// TIA Portal project "Proyecto" (V16)

(* hardware
DEVICE "S71500/ET200MP station_1"  S7-1500 station
   slot 0: "Perfil soporte_0"  Rack  6ES7 590-1***0-0AA0
   slot 1: "PLC_1"  CPU 1511-1 PN  6ES7 511-1AK01-0AB0  V2.8
      slot 3: "Display de la CPU_1"  6ES7591-1AA00-0AA0
      slot 32768: "Interfaz PROFINET_1"  X1
         slot 32769: "Puerto_1"  X1 P1
         slot 32770: "Puerto_2"  X1 P2
      slot 34817: "Virtual CP interface port_1"  Virtual CP interface port  Virtual CP interface port
DEVICE "S71500/ET200MP station_2"  S7-1500 station
   slot 0: "Perfil soporte_0"  Rack  6ES7 590-1***0-0AA0
   slot 1: "PLC_2"  CPU 1511-1 PN  6ES7 511-1AK01-0AB0  V2.8
      slot 3: "Display de la CPU_1"  6ES7591-1AA00-0AA0
      slot 32768: "Interfaz PROFINET_1"  X1
         slot 32769: "Puerto_1"  X1 P1
         slot 32770: "Puerto_2"  X1 P2
      slot 34817: "Virtual CP interface port_1"  Virtual CP interface port  Virtual CP interface port
*)

// ===== PLC "PLC_1"  CPU 1511-1 PN =====

VAR_GLOBAL   // PLC tag table "Tabla de variables estándar"
   "System_Byte" AT %MB1 : Byte;
   "FirstScan" AT %M1.0 : Bool;
   "DiagStatusUpdate" AT %M1.1 : Bool;
   "AlwaysTRUE" AT %M1.2 : Bool;
   "AlwaysFALSE" AT %M1.3 : Bool;
   "Clock_Byte" AT %MB0 : Byte;
   "Clock_10Hz" AT %M0.0 : Bool;
   "Clock_5Hz" AT %M0.1 : Bool;
   "Clock_2.5Hz" AT %M0.2 : Bool;
   "Clock_2Hz" AT %M0.3 : Bool;
   "Clock_1.25Hz" AT %M0.4 : Bool;
   "Clock_1Hz" AT %M0.5 : Bool;
   "Clock_0.625Hz" AT %M0.6 : Bool;
   "Clock_0.5Hz" AT %M0.7 : Bool;
END_VAR

DATA_BLOCK "DataLogPLC1Maestro"   // DB1
{ S7_Optimized_Access := 'FALSE' }
VERSION : 0.1
   VAR
      Variable1 : Real := 0.55;
      SetPoint : Int := 5;
   END_VAR
BEGIN
END_DATA_BLOCK

DATA_BLOCK "ProduccionPLC_Campo"   // DB4
{ S7_Optimized_Access := 'FALSE' }
VERSION : 0.1
   VAR
      Produccion : Array[1..7] of Real;
      EstadoMaquina : Array[1..2] of Bool;
   END_VAR
BEGIN
END_DATA_BLOCK

DATA_BLOCK "EnvioVariables"   // DB5
{ S7_Optimized_Access := 'FALSE' }
VERSION : 0.1
   VAR
      Variables : Array[1..8] of Bool;
   END_VAR
BEGIN
   Variables[1] := TRUE;
   Variables[2] := TRUE;
END_DATA_BLOCK

// folder: System blocks/Program resources

DATA_BLOCK "PLC_1_Receive_DB"   // DB2
{ S7_Optimized_Access := 'TRUE' }
AUTHOR : SIMATIC
FAMILY : MC7Plus
NAME : IP_RFC
VERSION : 1.0
// stored: InstanceOfName TCON_IP_RFC
"TCON_IP_RFC"
BEGIN
   ID := 1;
   InterfaceId := 64;
   LocalTSelector.TSel[1] := B#16#E0;
   LocalTSelector.TSel[2] := B#16#01;
   LocalTSelector.TSel[3] := B#16#49;
   LocalTSelector.TSel[4] := B#16#53;
   LocalTSelector.TSel[5] := B#16#4F;
   LocalTSelector.TSel[6] := B#16#6F;
   LocalTSelector.TSel[7] := B#16#6E;
   LocalTSelector.TSel[8] := B#16#54;
   LocalTSelector.TSel[9] := B#16#43;
   LocalTSelector.TSel[10] := B#16#50;
   LocalTSelector.TSel[11] := B#16#2D;
   LocalTSelector.TSel[12] := B#16#31;
   LocalTSelector.TSelLength := 12;
   RemoteTSelector.TSel[1] := B#16#E0;
   RemoteTSelector.TSel[2] := B#16#01;
   RemoteTSelector.TSel[3] := B#16#49;
   RemoteTSelector.TSel[4] := B#16#53;
   RemoteTSelector.TSel[5] := B#16#4F;
   RemoteTSelector.TSel[6] := B#16#6F;
   RemoteTSelector.TSel[7] := B#16#6E;
   RemoteTSelector.TSel[8] := B#16#54;
   RemoteTSelector.TSel[9] := B#16#43;
   RemoteTSelector.TSel[10] := B#16#50;
   RemoteTSelector.TSel[11] := B#16#2D;
   RemoteTSelector.TSel[12] := B#16#31;
   RemoteTSelector.TSelLength := 12;
   RemoteAddress.ADDR[1] := 192;
   RemoteAddress.ADDR[2] := 168;
   RemoteAddress.ADDR[4] := 41;
END_DATA_BLOCK

DATA_BLOCK "PLC_1_Send_DB"   // DB7
{ S7_Optimized_Access := 'TRUE' }
AUTHOR : SIMATIC
FAMILY : MC7Plus
NAME : IP_RFC
VERSION : 1.0
// stored: InstanceOfName TCON_IP_RFC
"TCON_IP_RFC"
BEGIN
   ID := 2;
   InterfaceId := 64;
   RemoteTSelector.TSel[1] := B#16#50;
   RemoteTSelector.TSel[2] := B#16#4C;
   RemoteTSelector.TSel[3] := B#16#43;
   RemoteTSelector.TSel[4] := B#16#32;
   RemoteTSelector.TSel[5] := B#16#5F;
   RemoteTSelector.TSel[6] := B#16#52;
   RemoteTSelector.TSel[7] := B#16#45;
   RemoteTSelector.TSel[8] := B#16#43;
   RemoteTSelector.TSel[9] := B#16#49;
   RemoteTSelector.TSel[10] := B#16#42;
   RemoteTSelector.TSel[11] := B#16#45;
   RemoteTSelector.TSelLength := 11;
   LocalTSelector.TSel[1] := B#16#50;
   LocalTSelector.TSel[2] := B#16#4C;
   LocalTSelector.TSel[3] := B#16#43;
   LocalTSelector.TSel[4] := B#16#31;
   LocalTSelector.TSel[5] := B#16#5F;
   LocalTSelector.TSel[6] := B#16#45;
   LocalTSelector.TSel[7] := B#16#4E;
   LocalTSelector.TSel[8] := B#16#56;
   LocalTSelector.TSel[9] := B#16#49;
   LocalTSelector.TSel[10] := B#16#41;
   LocalTSelector.TSelLength := 10;
   RemoteAddress.ADDR[1] := 192;
   RemoteAddress.ADDR[2] := 168;
   RemoteAddress.ADDR[4] := 41;
END_DATA_BLOCK

DATA_BLOCK "PLC_1_Receive_DB_1"   // DB8
{ S7_Optimized_Access := 'TRUE' }
AUTHOR : SIMATIC
FAMILY : MC7Plus
NAME : IP_RFC
VERSION : 1.0
// stored: InstanceOfName TCON_IP_RFC
"TCON_IP_RFC"
BEGIN
   ID := 3;
   InterfaceId := 64;
   LocalTSelector.TSel[1] := B#16#E0;
   LocalTSelector.TSel[2] := B#16#01;
   LocalTSelector.TSel[3] := B#16#49;
   LocalTSelector.TSel[4] := B#16#53;
   LocalTSelector.TSel[5] := B#16#4F;
   LocalTSelector.TSel[6] := B#16#6F;
   LocalTSelector.TSel[7] := B#16#6E;
   LocalTSelector.TSel[8] := B#16#54;
   LocalTSelector.TSel[9] := B#16#43;
   LocalTSelector.TSel[10] := B#16#50;
   LocalTSelector.TSel[11] := B#16#2D;
   LocalTSelector.TSel[12] := B#16#31;
   LocalTSelector.TSelLength := 12;
   RemoteTSelector.TSel[1] := B#16#E0;
   RemoteTSelector.TSel[2] := B#16#01;
   RemoteTSelector.TSel[3] := B#16#49;
   RemoteTSelector.TSel[4] := B#16#53;
   RemoteTSelector.TSel[5] := B#16#4F;
   RemoteTSelector.TSel[6] := B#16#6F;
   RemoteTSelector.TSel[7] := B#16#6E;
   RemoteTSelector.TSel[8] := B#16#54;
   RemoteTSelector.TSel[9] := B#16#43;
   RemoteTSelector.TSel[10] := B#16#50;
   RemoteTSelector.TSel[11] := B#16#2D;
   RemoteTSelector.TSel[12] := B#16#31;
   RemoteTSelector.TSelLength := 12;
   RemoteAddress.ADDR[1] := 192;
   RemoteAddress.ADDR[2] := 168;
   RemoteAddress.ADDR[4] := 41;
END_DATA_BLOCK

// folder: (top level)

FUNCTION "Generador_incremental" : Void   // FC1, SCL
{ S7_Optimized_Access := 'TRUE' }
VERSION : 0.1
   VAR_INPUT
      minimo : Real;
      maximo : Real;
      incremento : Real;
   END_VAR
   VAR_IN_OUT
      aleatorio : Real;
   END_VAR
BEGIN
   REGION Ajustar el valor minimo
       IF #aleatorio < #minimo THEN
           #aleatorio := #minimo;
       END_IF;
   END_REGION

   REGION Generador Incremental
       IF #aleatorio < #maximo THEN
           #aleatorio := #aleatorio + #incremento;
       ELSE
           #aleatorio := #minimo;
       END_IF;
   END_REGION
END_FUNCTION

FUNCTION "RecibirProduccion" : Void   // FC2, LAD
{ S7_Optimized_Access := 'TRUE' }
VERSION : 0.1
BEGIN

REGION Network 1
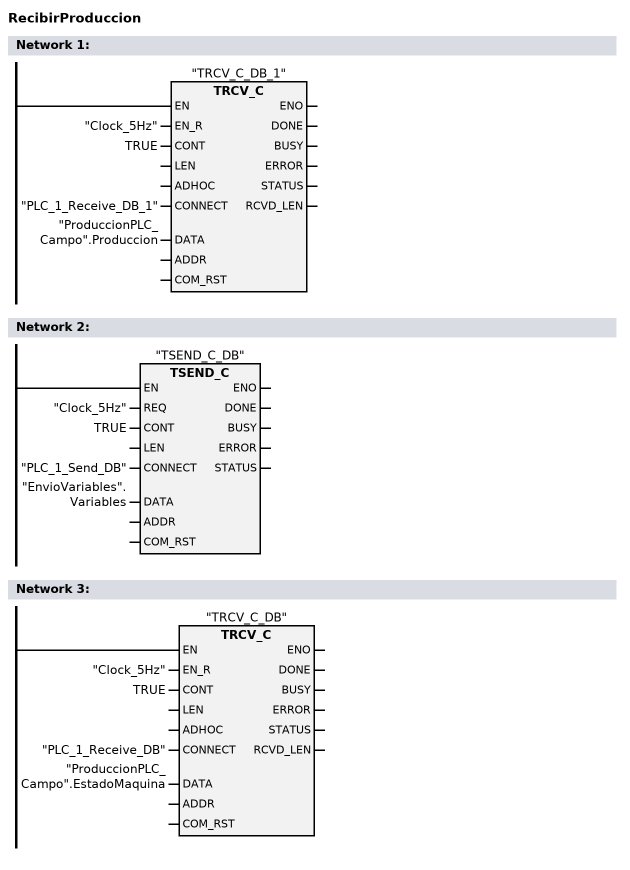
   "TRCV_C_DB_1"(EN_R := "Clock_5Hz",   // TRCV_C
                 CONT := TRUE,
                 CONNECT := "PLC_1_Receive_DB_1",
                 DATA := "ProduccionPLC_Campo".Produccion);
END_REGION

REGION Network 2
   "TSEND_C_DB"(REQ := "Clock_5Hz",   // TSEND_C
                CONT := TRUE,
                CONNECT := "PLC_1_Send_DB",
                DATA := "EnvioVariables".Variables);
END_REGION

REGION Network 3
   "TRCV_C_DB"(EN_R := "Clock_5Hz",   // TRCV_C
               CONT := TRUE,
               CONNECT := "PLC_1_Receive_DB",
               DATA := "ProduccionPLC_Campo".EstadoMaquina);
END_REGION
END_FUNCTION

ORGANIZATION_BLOCK "Main"   // OB1, LAD, ProgramCycle
TITLE = "Main Program Sweep (Cycle)"
{ S7_Optimized_Access := 'TRUE' }
VERSION : 0.1
   VAR_INPUT
      Initial_Call : Bool;   // Initial call of this OB
      Remanence : Bool;   // =True, if remanent data are available
   END_VAR
BEGIN

REGION Network 1
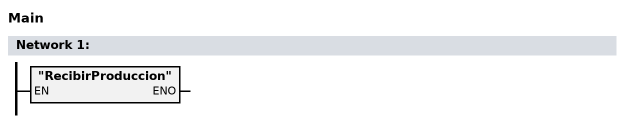
   RUNG wire#powerrail
      "RecibirProduccion"()
   END_RUNG
   // the same network as SCL:
   "RecibirProduccion"();
END_REGION
END_ORGANIZATION_BLOCK

// folder: LGF/4 Math operations

FUNCTION "LGF_RandomRange_Real" : Real   // FC10014, SCL
TITLE = LGF_RandomRange_Real
{ S7_Optimized_Access := 'TRUE' }
AUTHOR : Siemens_Digital_Industries
FAMILY : LGF
NAME : LGF_RandomRange_Real
// This function generates a random value in defined limits with each call.  
// The random number has the data type Real in the specified range.
// Diese Funktion generiert bei jedem Aufruf einen zufälligen Wert zwischen einem definierten Max- und Minwert.  
// Die Zufallszahl hat den Datentyp Real im spezifiziertem Wertebereich.
   VAR_INPUT
      minValue : Real;   // Minimalwert der für den Wertebereich der Zufallszahl - Untergrenze / Minimum value of the range of the random number - lower border
      maxValue : Real;   // Maximalwert der für den Wertebereich der Zufallszahl - Obergrenze / Maximum value of the range of the random number - upper border
   END_VAR
   VAR_OUTPUT
      error : Bool;   // FALSE: No error TRUE: An error occurred during the execution of the FB / FALSE: Kein Fehler TRUE: Während der Ausführung des FB ist ein Fehler aufgetreten
      status : Word;   // 16#0000-16#7FFF: Status of the FB 16#8000-16#FFFF: Error identification (see following Table) / 16#0000-16#7FFF: Status des FB 16#8000-16#FFFF: Fehleridentifikation (siehe folgende Tabelle)
      subfunctionStatus : Word;   // Status or return value of called FB's, FC's and system blocks / Status oder Rückgabewert von aufgerufenen FB's / FC's und Systemfunktionen
   END_VAR
   VAR_TEMP
      tempTime : DTL;   // Temp memory for System time / Temp variable für System Zeit
      tempNanoSecondInDWord : DWord;   // Temp UDInt converted to DWord for access to individual bytes / Temp UDInt konvertiert nach Dword für den Zufriff per Slice auf die Bytes
      tempTimeStatus : Word;   // Temp status of the instruction `RD_SYS_T` / Temp Status der Systemfunktion `RD_SYS_T`
      tempRandomValue : DWord;   // Temp Random startvalue / Temp Zufallswert als Startwert
      tempNormReal : Real;   // Temp normalized Real value (0.0 - 1.0) / Temp Normalisierer Realwert (0.0 - 1.0)
   END_VAR
   // Ret_Val : Random Real number in the predefined range / Zufallszahl vom Datentyp Real im definierten Wertebereich
   VAR CONSTANT
      ZERO : Real := 0.0;   // Zero / 0.0 - value in case of error / Null / 0.0 - Rückgabewert im Fehlerfall
      MAX_UDINT : UDInt := 4294967295;   // Maximum UDInt datatype / Maximalwert eines UDInt Datentype
      SUB_STATUS_NO_ERROR : Word := 16#0000;   // Status: sub function call ends without error / Status: Unterfunktionsaufruf ohne Fehler beendet
      STATUS_FINISHED_NO_ERROR : Word := 16#0000;   // Execution finished without errors / Abarbeitung ohne Fehler beendet
      ERR_MAX_LESS_MIN : Word := 16#8200;   // Error: The ranges specified are wrong: `minValue` is greater than `maxValue` / Fehler: Der spezifizierte Wetebereich is fehlerhaft: `minValue` ist größer als `maxValue`
      ERR_RD_SYS_T : Word := 16#8600;   // Error in `RD_SYS_T` command - check `subFunctionStatus` code / Fehler in Anweisung `RD_SYS_T` - weitere infos in `subFunctionStatus`
   END_VAR
BEGIN
   REGION Block info header
     //=============================================================================
     // SIEMENS AG / (c)Copyright 2017
     //-----------------------------------------------------------------------------
     // Title:            LGF_RandomRange_Real
     // Comment/Function: This function generates random numbers in defined limits (Datatype Real)
     // Library/Family:   LGF(Library General Functions)
     // Author:           Siemens Digital Industry Support
     // Tested with:      S7-PLCSIM Advanced V2.0 SP1
     // Engineering:      TIA Portal V15 Update 2
     // Restrictions:     ENO disabled - error handling done by error and status
     // Requirements:     PLC (S7-1200 / S7-1500)
     //-------------------------------------------------------------------------------
     // Change log table:
     // Version  | Date       | Expert in charge       | Changes applied
     //----------|------------|------------------------|------------------------------
     // 01.00.00 19.08.2015  Siemens Industry Online Support
     //                      First released version
     // 01.00.01 02.01.2017  Siemens Industry Online Support
     //                      Upgrade: TIA Portal V14 Update 1
     // 01.00.02 02.03.2017  Siemens Industry Online Support
     //                      Bugfix: FC number
     // 01.00.03 17.08.2018  Siemens Industry Online Support
     //                      Upgrade: TIA V15 Update 2
     // 01.00.04 23.11.2018  Siemens Industry Online Support
     //                      Upgrade: TIA V15.1
     // 01.01.00 13.11.2019  Simatic Systems Support
     //                      Renamed from "LGF_RandomReal" to "LGF_RandomRange_Real"
     //                      Regions, comments and constants are added
     // 03.00.00 23.04.2020  Simatic Systems Support
     //                      Set version to V3.0.0, harmonize the version of the whole library
     // 03.00.01 04.02.2021  Simatic Systems Support
     //                      Insert documentation
     //=============================================================================
   END_REGION Block info header

   REGION DESCRIPTION
     (/*Note
   :    The status of called commands is output in `subFunctionStatus`. In this case, the output value in `status` indicates which command caused the error. In this case, refer to the TIA Portal Online Help section for information on the respective commands.

   The block generates random values that are between the specified `minValue` and the `maxValue`. This random value is output via the `Ret_Val`.

   The random value is formed from the nanoseconds of the current system time of the CPU. The byte order of this value is inverted and then converted to a floating point.
   Hinweis
   :    In `subFunctionStatus` wird der Status von aufgerufenen Anweisungen ausgegeben. Der Ausgangswert in `status` gibt in diesem Fall an, welche Anweisung den Fehler verursacht hat. Holen Sie sich in diesem Fall die Informationen aus der TIA Portal Online Hilfe zu den jeweiligen Anweisungen.

   Der Baustein generiert zufällige Werte, die zwischen dem angegebenen `minValue`-Wert und `maxValue`-Wert liegen. Dieser zufällige Wert wird über den `Ret_Val` ausgegeben.

   Der Zufallswert wird aus den Nanosekunden der aktuellen Systemzeit der CPU gebildet. Dabei wird die Bytereihenfolge dieses Wertes invertiert und anschließend in eine Gleitkommazahl ungewandelt.*/)
   END_REGION DESCRIPTION

   REGION Validation
     // Check if the maximal Value is less than the minimal value
     IF (#minValue > #maxValue) THEN
       #error := true;
       #status := #ERR_MAX_LESS_MIN;
       #subfunctionStatus := #SUB_STATUS_NO_ERROR;
       #LGF_RandomRange_Real := #ZERO;
       RETURN;
     END_IF;

     // Read system time
     #tempTimeStatus := INT_TO_WORD(RD_SYS_T(#tempTime));

     // Check return variable for error
     IF (#tempTimeStatus <> #SUB_STATUS_NO_ERROR) THEN
       #error := true;
       #status := #ERR_RD_SYS_T;
       #subfunctionStatus := #tempTimeStatus;
       #LGF_RandomRange_Real := #ZERO;
       RETURN;
     END_IF;
   END_REGION

   REGION Calculating random number
     // Converting to double word so individual bytes can be addressed
     #tempNanoSecondInDWord := UDINT_TO_DWORD(#tempTime.NANOSECOND);

     // Calculate a random-start-value depending on the time
     #tempRandomValue.%B3 := #tempNanoSecondInDWord.%B0;
     #tempRandomValue.%B2 := #tempNanoSecondInDWord.%B1;
     #tempRandomValue.%B1 := #tempNanoSecondInDWord.%B2;
     #tempRandomValue.%B0 := #tempNanoSecondInDWord.%B3;

     // Norm the calculated random number: 0.0 <= #tempNormReal <= 1.0
     #tempNormReal := UDINT_TO_REAL(DWORD_TO_UDINT(#tempRandomValue)) / UDINT_TO_REAL(#MAX_UDINT);

     // Scale the tempNormReal to be in the range of maxValue and minValue
     #LGF_RandomRange_Real := ((#tempNormReal * (#maxValue - #minValue) + (#minValue)));

     #error := false;
     #status := #STATUS_FINISHED_NO_ERROR;
     #subfunctionStatus := #SUB_STATUS_NO_ERROR;
     // ENO mechanism is not used
     ENO := TRUE;
   END_REGION
END_FUNCTION

// ===== PLC "PLC_2"  CPU 1511-1 PN =====

VAR_GLOBAL   // PLC tag table "Tabla de variables estándar"
   "System_Byte" AT %MB1 : Byte;
   "FirstScan" AT %M1.0 : Bool;
   "DiagStatusUpdate" AT %M1.1 : Bool;
   "AlwaysTRUE" AT %M1.2 : Bool;
   "AlwaysFALSE" AT %M1.3 : Bool;
   "Clock_Byte" AT %MB0 : Byte;
   "Clock_10Hz" AT %M0.0 : Bool;
   "Clock_5Hz" AT %M0.1 : Bool;
   "Clock_2.5Hz" AT %M0.2 : Bool;
   "Clock_2Hz" AT %M0.3 : Bool;
   "Clock_1.25Hz" AT %M0.4 : Bool;
   "Clock_1Hz" AT %M0.5 : Bool;
   "Clock_0.625Hz" AT %M0.6 : Bool;
   "Clock_0.5Hz" AT %M0.7 : Bool;
   "Start" AT %I1.2 : Bool;
   "PASO0" AT %M10.3 : Bool;
   "PASO1" AT %M10.4 : Bool;
   "PASO2" AT %M10.5 : Bool;
   "PASO3" AT %M10.6 : Bool;
   "PASO4" AT %M10.7 : Bool;
   "PASO5" AT %M11.0 : Bool;
   "PASO6" AT %M11.1 : Bool;
   "PASO7" AT %M11.2 : Bool;
   "PASO8" AT %M11.3 : Bool;
   "PASO9" AT %M11.4 : Bool;
   "Motor_bases" AT %Q0.3 : Bool;
   "Motor_tapas" AT %Q0.6 : Bool;
   "Detector_bases" AT %I0.3 : Bool;
   "Detector_tapas" AT %I0.6 : Bool;
   "Presionar_bases" AT %Q0.4 : Bool;
   "Presionar_tapas" AT %Q0.7 : Bool;
   "MoverZ" AT %Q0.1 : Bool;
   "MoverX" AT %Q0.0 : Bool;
   "Agarrar" AT %Q0.2 : Bool;
   "MoviendoseZ" AT %I0.1 : Bool;
   "ItemDetectado" AT %I0.2 : Bool;
   "MoviendoseX" AT %I0.0 : Bool;
   "Base_posicionada" AT %I0.4 : Bool;
   "Tapa_posicionada" AT %I0.7 : Bool;
   "PASO10" AT %M11.5 : Bool;
   "PASO11" AT %M12.0 : Bool;
   "PASO12" AT %M12.1 : Bool;
   "PASO13" AT %M12.2 : Bool;
   "PASO14" AT %M12.3 : Bool;
   "PASO15" AT %M12.4 : Bool;
   "PASO16" AT %M12.5 : Bool;
   "PASO17" AT %M12.6 : Bool;
   "PASO18" AT %M12.7 : Bool;
   "Libera_base" AT %Q1.0 : Bool;
   "Saliendo" AT %I1.1 : Bool;
   "PASO9_INTER" AT %M2.0 : Bool;
   "PASO2_INTER" AT %M2.1 : Bool;
   "PASO2_INTER2" AT %M2.2 : Bool;
   "Done" AT %M2.3 : Bool;
   "EmisorBases" AT %Q1.4 : Bool;
   "EmisorTapas" AT %Q1.5 : Bool;
   "SP_Cajas" AT %MW4 : Int;
   "SP_CajasAUX" AT %MW6 : Int;
   "RESET_COUNTER" AT %M2.4 : Bool;
   "PASO9_INTER2" AT %M2.5 : Bool;
   "SetPointInterno" AT %MW8 : Int;
   "Stop" AT %I1.4 : Bool;
   "AUX1" AT %M2.6 : Bool;
   "AUX2" AT %M2.7 : Bool;
   "AUX3" AT %M3.0 : Bool;
   "SET DETEC" AT %M3.1 : Bool;
   "Sensor tapa" AT %ID100 : DInt;
   "Sensor base" AT %ID104 : DInt;
   "Reset" AT %I1.3 : Bool;
   "Emergency stop" AT %I1.5 : Bool;
   "RESET_DONE" AT %M3.2 : Bool;
   "TiempoMinutos" AT %MD14 : Real;
   "FactoryRunning" AT %I1.7 : Bool;
   "TiempoTotal" AT %MD18 : Real;
   "Div1" AT %MD22 : Real;
END_VAR

DATA_BLOCK "Datalog"   // DB1
{ S7_Optimized_Access := 'FALSE' }
VERSION : 0.1
   VAR
      Variable1 : Real;
      SetPoint : Int := 4;
   END_VAR
BEGIN
END_DATA_BLOCK

DATA_BLOCK "Envio_Estados"   // DB12
{ S7_Optimized_Access := 'TRUE' }
VERSION : 0.1
   VAR
      Parametros : Array[1..7] of Real;
      EstadoMaquina : Array[1..2] of Bool;
   END_VAR
BEGIN
END_DATA_BLOCK

DATA_BLOCK "RecepcionVariables"   // DB17
{ S7_Optimized_Access := 'TRUE' }
VERSION : 0.1
   VAR
      Variables : Array[1..8] of Bool;
   END_VAR
BEGIN
END_DATA_BLOCK

// folder: System blocks/Program resources

DATA_BLOCK "IEC_Timer_0_DB"   // DB2
{ S7_Optimized_Access := 'TRUE' }
AUTHOR : Simatic
FAMILY : IEC
NAME : IEC_TMR
VERSION : 1.0
// stored: InstanceOfName IEC_TIMER
"IEC_TIMER"
BEGIN
END_DATA_BLOCK

DATA_BLOCK "IEC_Timer_0_DB_1"   // DB3
{ S7_Optimized_Access := 'TRUE' }
AUTHOR : Simatic
FAMILY : IEC
NAME : IEC_TMR
VERSION : 1.0
// stored: InstanceOfName IEC_TIMER
"IEC_TIMER"
BEGIN
END_DATA_BLOCK

DATA_BLOCK "IEC_Timer_0_DB_2"   // DB4
{ S7_Optimized_Access := 'TRUE' }
AUTHOR : Simatic
FAMILY : IEC
NAME : IEC_TMR
VERSION : 1.0
// stored: InstanceOfName IEC_TIMER
"IEC_TIMER"
BEGIN
END_DATA_BLOCK

DATA_BLOCK "IEC_Timer_0_DB_3"   // DB5
{ S7_Optimized_Access := 'TRUE' }
AUTHOR : Simatic
FAMILY : IEC
NAME : IEC_TMR
VERSION : 1.0
// stored: InstanceOfName IEC_TIMER
"IEC_TIMER"
BEGIN
END_DATA_BLOCK

DATA_BLOCK "IEC_Timer_0_DB_4"   // DB6
{ S7_Optimized_Access := 'TRUE' }
AUTHOR : Simatic
FAMILY : IEC
NAME : IEC_TMR
VERSION : 1.0
// stored: InstanceOfName IEC_TIMER
"IEC_TIMER"
BEGIN
END_DATA_BLOCK

DATA_BLOCK "IEC_Timer_0_DB_5"   // DB7
{ S7_Optimized_Access := 'TRUE' }
AUTHOR : Simatic
FAMILY : IEC
NAME : IEC_TMR
VERSION : 1.0
// stored: InstanceOfName IEC_TIMER
"IEC_TIMER"
BEGIN
END_DATA_BLOCK

DATA_BLOCK "IEC_Timer_0_DB_6"   // DB8
{ S7_Optimized_Access := 'TRUE' }
AUTHOR : Simatic
FAMILY : IEC
NAME : IEC_TMR
VERSION : 1.0
// stored: InstanceOfName IEC_TIMER
"IEC_TIMER"
BEGIN
END_DATA_BLOCK

DATA_BLOCK "IEC_Counter_0_DB"   // DB9
{ S7_Optimized_Access := 'TRUE' }
AUTHOR : Simatic
FAMILY : IEC
NAME : CNTR
VERSION : 1.0
// stored: InstanceOfName IEC_COUNTER
"IEC_COUNTER"
BEGIN
END_DATA_BLOCK

DATA_BLOCK "IEC_Timer_0_DB_8"   // DB10
{ S7_Optimized_Access := 'TRUE' }
AUTHOR : Simatic
FAMILY : IEC
NAME : IEC_TMR
VERSION : 1.0
// stored: InstanceOfName IEC_TIMER
"IEC_TIMER"
BEGIN
END_DATA_BLOCK

DATA_BLOCK "IEC_Timer_0_DB_7"   // DB11
{ S7_Optimized_Access := 'TRUE' }
AUTHOR : Simatic
FAMILY : IEC
NAME : IEC_TMR
VERSION : 1.0
// stored: InstanceOfName IEC_TIMER
"IEC_TIMER"
BEGIN
END_DATA_BLOCK

DATA_BLOCK "PLC_2_Send_DB"   // DB15
{ S7_Optimized_Access := 'TRUE' }
AUTHOR : SIMATIC
FAMILY : MC7Plus
NAME : IP_RFC
VERSION : 1.0
// stored: InstanceOfName TCON_IP_RFC
"TCON_IP_RFC"
BEGIN
   ID := 1;
   ActiveEstablished := true;
   InterfaceId := 64;
   RemoteAddress.ADDR[1] := 192;
   RemoteAddress.ADDR[2] := 168;
   RemoteAddress.ADDR[4] := 21;
   LocalTSelector.TSel[1] := B#16#E0;
   LocalTSelector.TSel[2] := B#16#01;
   LocalTSelector.TSel[3] := B#16#49;
   LocalTSelector.TSel[4] := B#16#53;
   LocalTSelector.TSel[5] := B#16#4F;
   LocalTSelector.TSel[6] := B#16#6F;
   LocalTSelector.TSel[7] := B#16#6E;
   LocalTSelector.TSel[8] := B#16#54;
   LocalTSelector.TSel[9] := B#16#43;
   LocalTSelector.TSel[10] := B#16#50;
   LocalTSelector.TSel[11] := B#16#2D;
   LocalTSelector.TSel[12] := B#16#31;
   LocalTSelector.TSelLength := 12;
   RemoteTSelector.TSel[1] := B#16#E0;
   RemoteTSelector.TSel[2] := B#16#01;
   RemoteTSelector.TSel[3] := B#16#49;
   RemoteTSelector.TSel[4] := B#16#53;
   RemoteTSelector.TSel[5] := B#16#4F;
   RemoteTSelector.TSel[6] := B#16#6F;
   RemoteTSelector.TSel[7] := B#16#6E;
   RemoteTSelector.TSel[8] := B#16#54;
   RemoteTSelector.TSel[9] := B#16#43;
   RemoteTSelector.TSel[10] := B#16#50;
   RemoteTSelector.TSel[11] := B#16#2D;
   RemoteTSelector.TSel[12] := B#16#31;
   RemoteTSelector.TSelLength := 12;
END_DATA_BLOCK

DATA_BLOCK "PLC_2_Receive_DB"   // DB16
{ S7_Optimized_Access := 'TRUE' }
AUTHOR : SIMATIC
FAMILY : MC7Plus
NAME : IP_RFC
VERSION : 1.0
// stored: InstanceOfName TCON_IP_RFC
"TCON_IP_RFC"
BEGIN
   ID := 2;
   ActiveEstablished := true;
   InterfaceId := 64;
   RemoteAddress.ADDR[1] := 192;
   RemoteAddress.ADDR[2] := 168;
   RemoteAddress.ADDR[4] := 21;
   LocalTSelector.TSel[1] := B#16#50;
   LocalTSelector.TSel[2] := B#16#4C;
   LocalTSelector.TSel[3] := B#16#43;
   LocalTSelector.TSel[4] := B#16#32;
   LocalTSelector.TSel[5] := B#16#5F;
   LocalTSelector.TSel[6] := B#16#52;
   LocalTSelector.TSel[7] := B#16#45;
   LocalTSelector.TSel[8] := B#16#43;
   LocalTSelector.TSel[9] := B#16#49;
   LocalTSelector.TSel[10] := B#16#42;
   LocalTSelector.TSel[11] := B#16#45;
   LocalTSelector.TSelLength := 11;
   RemoteTSelector.TSel[1] := B#16#50;
   RemoteTSelector.TSel[2] := B#16#4C;
   RemoteTSelector.TSel[3] := B#16#43;
   RemoteTSelector.TSel[4] := B#16#31;
   RemoteTSelector.TSel[5] := B#16#5F;
   RemoteTSelector.TSel[6] := B#16#45;
   RemoteTSelector.TSel[7] := B#16#4E;
   RemoteTSelector.TSel[8] := B#16#56;
   RemoteTSelector.TSel[9] := B#16#49;
   RemoteTSelector.TSel[10] := B#16#41;
   RemoteTSelector.TSelLength := 10;
END_DATA_BLOCK

DATA_BLOCK "Tipo1VV"   // DB19
{ S7_Optimized_Access := 'TRUE' }
AUTHOR : Simatic
FAMILY : IEC
NAME : CNTR
VERSION : 1.0
// stored: InstanceOfName IEC_COUNTER
"IEC_COUNTER"
BEGIN
END_DATA_BLOCK

DATA_BLOCK "IEC_Timer_0_DB_10"   // DB20
{ S7_Optimized_Access := 'TRUE' }
AUTHOR : Simatic
FAMILY : IEC
NAME : IEC_TMR
VERSION : 1.0
// stored: InstanceOfName IEC_TIMER
"IEC_TIMER"
BEGIN
END_DATA_BLOCK

DATA_BLOCK "IEC_Timer_0_DB_11"   // DB21
{ S7_Optimized_Access := 'TRUE' }
AUTHOR : Simatic
FAMILY : IEC
NAME : IEC_TMR
VERSION : 1.0
// stored: InstanceOfName IEC_TIMER
"IEC_TIMER"
BEGIN
END_DATA_BLOCK

DATA_BLOCK "Tipo1VA"   // DB22
{ S7_Optimized_Access := 'TRUE' }
AUTHOR : Simatic
FAMILY : IEC
NAME : CNTR
VERSION : 1.0
// stored: InstanceOfName IEC_COUNTER
"IEC_COUNTER"
BEGIN
END_DATA_BLOCK

DATA_BLOCK "Tipo1AV"   // DB23
{ S7_Optimized_Access := 'TRUE' }
AUTHOR : Simatic
FAMILY : IEC
NAME : CNTR
VERSION : 1.0
// stored: InstanceOfName IEC_COUNTER
"IEC_COUNTER"
BEGIN
END_DATA_BLOCK

DATA_BLOCK "Tipo1AA"   // DB24
{ S7_Optimized_Access := 'TRUE' }
AUTHOR : Simatic
FAMILY : IEC
NAME : CNTR
VERSION : 1.0
// stored: InstanceOfName IEC_COUNTER
"IEC_COUNTER"
BEGIN
END_DATA_BLOCK

DATA_BLOCK "IEC_Counter_0_DB_1"   // DB25
{ S7_Optimized_Access := 'TRUE' }
AUTHOR : Simatic
FAMILY : IEC
NAME : CNTR
VERSION : 1.0
// stored: InstanceOfName IEC_COUNTER
"IEC_COUNTER"
BEGIN
END_DATA_BLOCK

DATA_BLOCK "IEC_Counter_0_DB_2"   // DB26
{ S7_Optimized_Access := 'TRUE' }
AUTHOR : Simatic
FAMILY : IEC
NAME : CNTR
VERSION : 1.0
// stored: InstanceOfName IEC_COUNTER
"IEC_COUNTER"
BEGIN
END_DATA_BLOCK

DATA_BLOCK "IEC_Counter_0_DB_3"   // DB27
{ S7_Optimized_Access := 'TRUE' }
AUTHOR : Simatic
FAMILY : IEC
NAME : CNTR
VERSION : 1.0
// stored: InstanceOfName IEC_COUNTER
"IEC_COUNTER"
BEGIN
END_DATA_BLOCK

DATA_BLOCK "PLC_2_Send_DB_1"   // DB29
{ S7_Optimized_Access := 'TRUE' }
AUTHOR : SIMATIC
FAMILY : MC7Plus
NAME : IP_RFC
VERSION : 1.0
// stored: InstanceOfName TCON_IP_RFC
"TCON_IP_RFC"
BEGIN
   ID := 3;
   ActiveEstablished := true;
   InterfaceId := 64;
   RemoteAddress.ADDR[1] := 192;
   RemoteAddress.ADDR[2] := 168;
   RemoteAddress.ADDR[4] := 21;
   LocalTSelector.TSel[1] := B#16#E0;
   LocalTSelector.TSel[2] := B#16#01;
   LocalTSelector.TSel[3] := B#16#49;
   LocalTSelector.TSel[4] := B#16#53;
   LocalTSelector.TSel[5] := B#16#4F;
   LocalTSelector.TSel[6] := B#16#6F;
   LocalTSelector.TSel[7] := B#16#6E;
   LocalTSelector.TSel[8] := B#16#54;
   LocalTSelector.TSel[9] := B#16#43;
   LocalTSelector.TSel[10] := B#16#50;
   LocalTSelector.TSel[11] := B#16#2D;
   LocalTSelector.TSel[12] := B#16#31;
   LocalTSelector.TSelLength := 12;
   RemoteTSelector.TSel[1] := B#16#E0;
   RemoteTSelector.TSel[2] := B#16#01;
   RemoteTSelector.TSel[3] := B#16#49;
   RemoteTSelector.TSel[4] := B#16#53;
   RemoteTSelector.TSel[5] := B#16#4F;
   RemoteTSelector.TSel[6] := B#16#6F;
   RemoteTSelector.TSel[7] := B#16#6E;
   RemoteTSelector.TSel[8] := B#16#54;
   RemoteTSelector.TSel[9] := B#16#43;
   RemoteTSelector.TSel[10] := B#16#50;
   RemoteTSelector.TSel[11] := B#16#2D;
   RemoteTSelector.TSel[12] := B#16#31;
   RemoteTSelector.TSelLength := 12;
END_DATA_BLOCK

// folder: (top level)

FUNCTION "Envio_Datps" : Void   // FC1, LAD
{ S7_Optimized_Access := 'TRUE' }
VERSION : 0.1
BEGIN

REGION Network 1
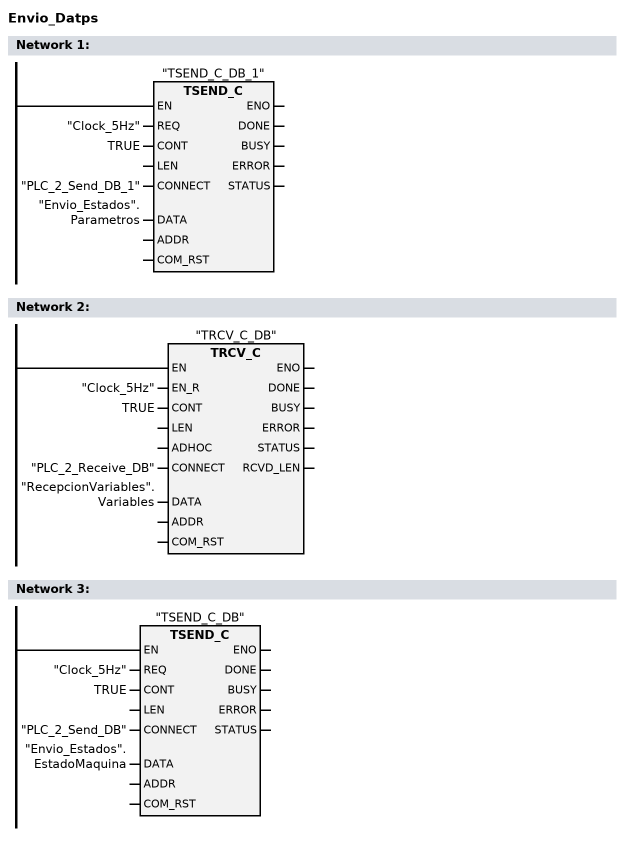
   "TSEND_C_DB_1"(REQ := "Clock_5Hz",   // TSEND_C
                  CONT := TRUE,
                  CONNECT := "PLC_2_Send_DB_1",
                  DATA := "Envio_Estados".Parametros);
END_REGION

REGION Network 2
   "TRCV_C_DB"(EN_R := "Clock_5Hz",   // TRCV_C
               CONT := TRUE,
               CONNECT := "PLC_2_Receive_DB",
               DATA := "RecepcionVariables".Variables);
END_REGION

REGION Network 3
   "TSEND_C_DB"(REQ := "Clock_5Hz",   // TSEND_C
                CONT := TRUE,
                CONNECT := "PLC_2_Send_DB",
                DATA := "Envio_Estados".EstadoMaquina);
END_REGION
END_FUNCTION

FUNCTION "RecepcionarDatos" : Void   // FC2, LAD
{ S7_Optimized_Access := 'TRUE' }
VERSION : 0.1
BEGIN

REGION Network 1
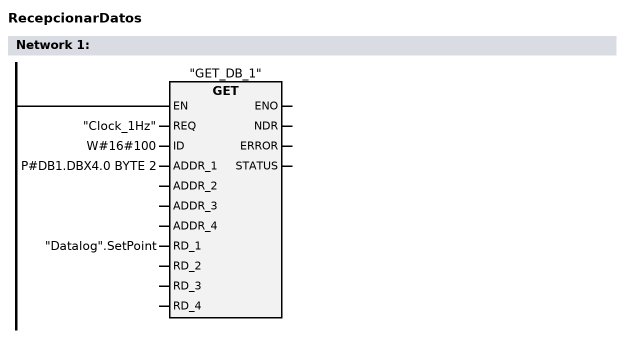
   "GET_DB_1"(REQ := "Clock_1Hz", ID := W#16#100, ADDR_1 := P#DB1.DBX4.0 BYTE 2, RD_1 := "Datalog".SetPoint);   // GET
END_REGION
END_FUNCTION

ORGANIZATION_BLOCK "Main"   // OB1, LAD, ProgramCycle
TITLE = "Main Program Sweep (Cycle)"
{ S7_Optimized_Access := 'TRUE' }
VERSION : 0.1
   VAR_INPUT
      Initial_Call : Bool;   // Initial call of this OB
      Remanence : Bool;   // =True, if remanent data are available
   END_VAR
   VAR_TEMP
      contador1 : Int;
      contador2 : Int;
      contador3 : Int;
      contador4 : Int;
   END_VAR
   VAR_TEMP   // added for the SCL form of the ladder/FBD networks
      _w1 : Bool;
      _w2 : Bool;
   END_VAR
BEGIN

REGION Network 1
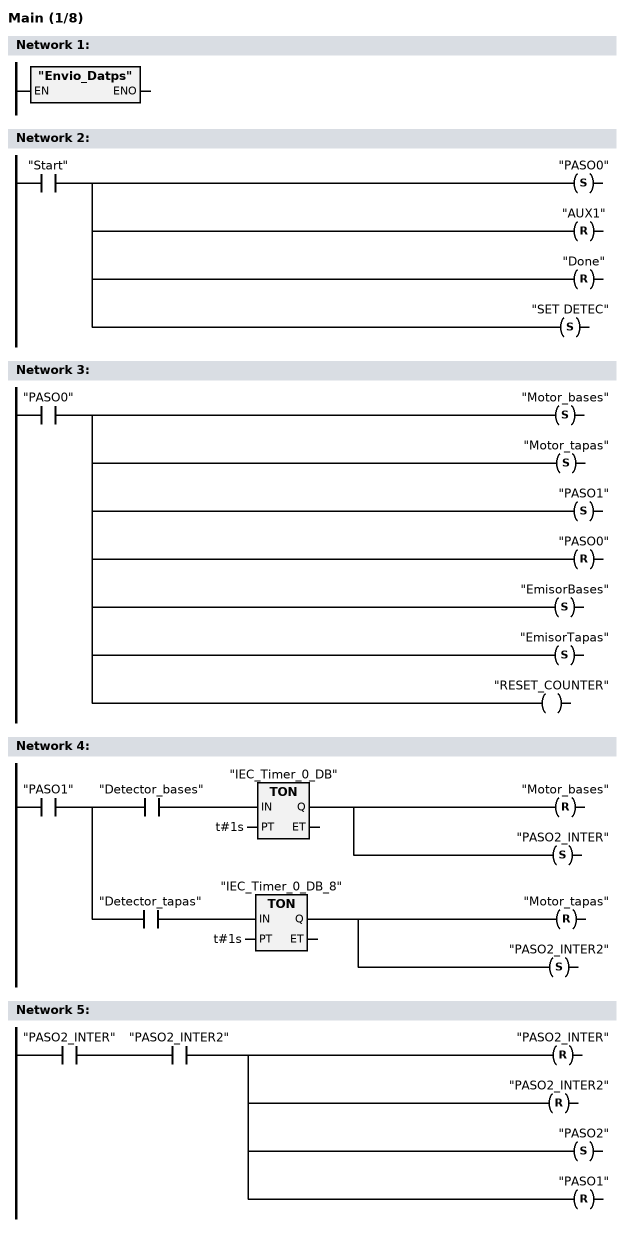
   RUNG wire#powerrail
      "Envio_Datps"()
   END_RUNG
   // the same network as SCL:
   "Envio_Datps"();
END_REGION

REGION Network 2
   RUNG wire#powerrail
      Contact( "Start" )
      wire#w1
      S_Coil( "PASO0" )
   END_RUNG
   RUNG wire#w1
      R_Coil( "AUX1" )
   END_RUNG
   RUNG wire#w1
      R_Coil( "Done" )
   END_RUNG
   RUNG wire#w1
      S_Coil( "SET DETEC" )
   END_RUNG
   // the same network as SCL:
   IF "Start" THEN
       "PASO0" := TRUE;
       "AUX1" := FALSE;
       "Done" := FALSE;
       "SET DETEC" := TRUE;
   END_IF;
END_REGION

REGION Network 3
   RUNG wire#powerrail
      Contact( "PASO0" )
      wire#w1
      S_Coil( "Motor_bases" )
   END_RUNG
   RUNG wire#w1
      S_Coil( "Motor_tapas" )
   END_RUNG
   RUNG wire#w1
      S_Coil( "PASO1" )
   END_RUNG
   RUNG wire#w1
      R_Coil( "PASO0" )
   END_RUNG
   RUNG wire#w1
      S_Coil( "EmisorBases" )
   END_RUNG
   RUNG wire#w1
      S_Coil( "EmisorTapas" )
   END_RUNG
   RUNG wire#w1
      Coil( "RESET_COUNTER" )
   END_RUNG
   // the same network as SCL:
   IF "PASO0" THEN
       "Motor_bases" := TRUE;
       "Motor_tapas" := TRUE;
       "PASO1" := TRUE;
   END_IF;
   #_w1 := "PASO0";
   IF #_w1 THEN
       "PASO0" := FALSE;
       "EmisorBases" := TRUE;
       "EmisorTapas" := TRUE;
   END_IF;
   "RESET_COUNTER" := #_w1;
END_REGION

REGION Network 4
   "IEC_Timer_0_DB".TON(IN := "PASO1" AND "Detector_bases", PT := t#1s);
   IF "IEC_Timer_0_DB".Q THEN
       "Motor_bases" := FALSE;
       "PASO2_INTER" := TRUE;
   END_IF;
   "IEC_Timer_0_DB_8".TON(IN := "PASO1" AND "Detector_tapas", PT := t#1s);
   IF "IEC_Timer_0_DB_8".Q THEN
       "Motor_tapas" := FALSE;
       "PASO2_INTER2" := TRUE;
   END_IF;
END_REGION

REGION Network 5
   RUNG wire#powerrail
      Contact( "PASO2_INTER" )
      Contact( "PASO2_INTER2" )
      wire#w1
      R_Coil( "PASO2_INTER" )
   END_RUNG
   RUNG wire#w1
      R_Coil( "PASO2_INTER2" )
   END_RUNG
   RUNG wire#w1
      S_Coil( "PASO2" )
   END_RUNG
   RUNG wire#w1
      R_Coil( "PASO1" )
   END_RUNG
   // the same network as SCL:
   #_w1 := "PASO2_INTER" AND "PASO2_INTER2";
   IF #_w1 THEN
       "PASO2_INTER" := FALSE;
       "PASO2_INTER2" := FALSE;
       "PASO2" := TRUE;
       "PASO1" := FALSE;
   END_IF;
END_REGION

REGION Network 6
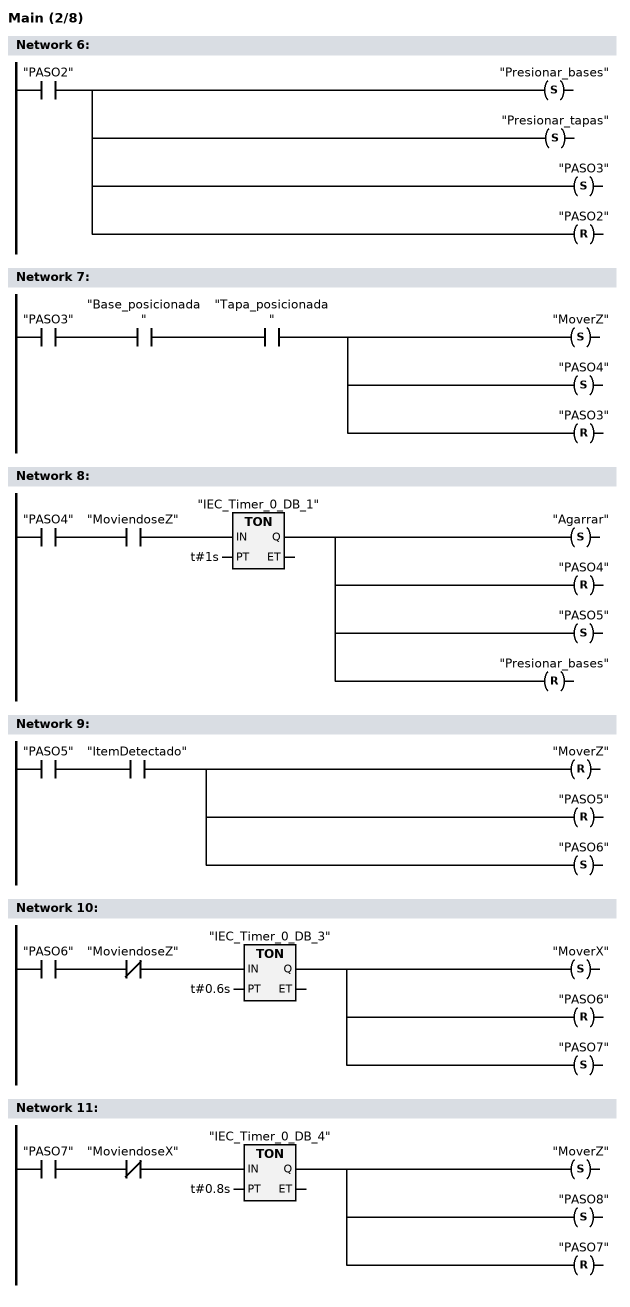
   RUNG wire#powerrail
      Contact( "PASO2" )
      wire#w1
      S_Coil( "Presionar_bases" )
   END_RUNG
   RUNG wire#w1
      S_Coil( "Presionar_tapas" )
   END_RUNG
   RUNG wire#w1
      S_Coil( "PASO3" )
   END_RUNG
   RUNG wire#w1
      R_Coil( "PASO2" )
   END_RUNG
   // the same network as SCL:
   IF "PASO2" THEN
       "Presionar_bases" := TRUE;
       "Presionar_tapas" := TRUE;
       "PASO3" := TRUE;
       "PASO2" := FALSE;
   END_IF;
END_REGION

REGION Network 7
   RUNG wire#powerrail
      Contact( "PASO3" )
      Contact( "Base_posicionada" )
      Contact( "Tapa_posicionada" )
      wire#w1
      S_Coil( "MoverZ" )
   END_RUNG
   RUNG wire#w1
      S_Coil( "PASO4" )
   END_RUNG
   RUNG wire#w1
      R_Coil( "PASO3" )
   END_RUNG
   // the same network as SCL:
   IF "PASO3" AND "Base_posicionada" AND "Tapa_posicionada" THEN
       "MoverZ" := TRUE;
       "PASO4" := TRUE;
       "PASO3" := FALSE;
   END_IF;
END_REGION

REGION Network 8
   "IEC_Timer_0_DB_1".TON(IN := "PASO4" AND "MoviendoseZ", PT := t#1s);
   IF "IEC_Timer_0_DB_1".Q THEN
       "Agarrar" := TRUE;
       "PASO4" := FALSE;
       "PASO5" := TRUE;
       "Presionar_bases" := FALSE;
   END_IF;
END_REGION

REGION Network 9
   RUNG wire#powerrail
      Contact( "PASO5" )
      Contact( "ItemDetectado" )
      wire#w1
      R_Coil( "MoverZ" )
   END_RUNG
   RUNG wire#w1
      R_Coil( "PASO5" )
   END_RUNG
   RUNG wire#w1
      S_Coil( "PASO6" )
   END_RUNG
   // the same network as SCL:
   IF "PASO5" AND "ItemDetectado" THEN "MoverZ" := FALSE; END_IF;
   #_w1 := "PASO5" AND "ItemDetectado";
   IF #_w1 THEN
       "PASO5" := FALSE;
       "PASO6" := TRUE;
   END_IF;
END_REGION

REGION Network 10
   "IEC_Timer_0_DB_3".TON(IN := "PASO6" AND NOT "MoviendoseZ", PT := t#0.6s);
   IF "IEC_Timer_0_DB_3".Q THEN
       "MoverX" := TRUE;
       "PASO6" := FALSE;
       "PASO7" := TRUE;
   END_IF;
END_REGION

REGION Network 11
   "IEC_Timer_0_DB_4".TON(IN := "PASO7" AND NOT "MoviendoseX", PT := t#0.8s);
   IF "IEC_Timer_0_DB_4".Q THEN
       "MoverZ" := TRUE;
       "PASO8" := TRUE;
       "PASO7" := FALSE;
   END_IF;
END_REGION

REGION Network 12
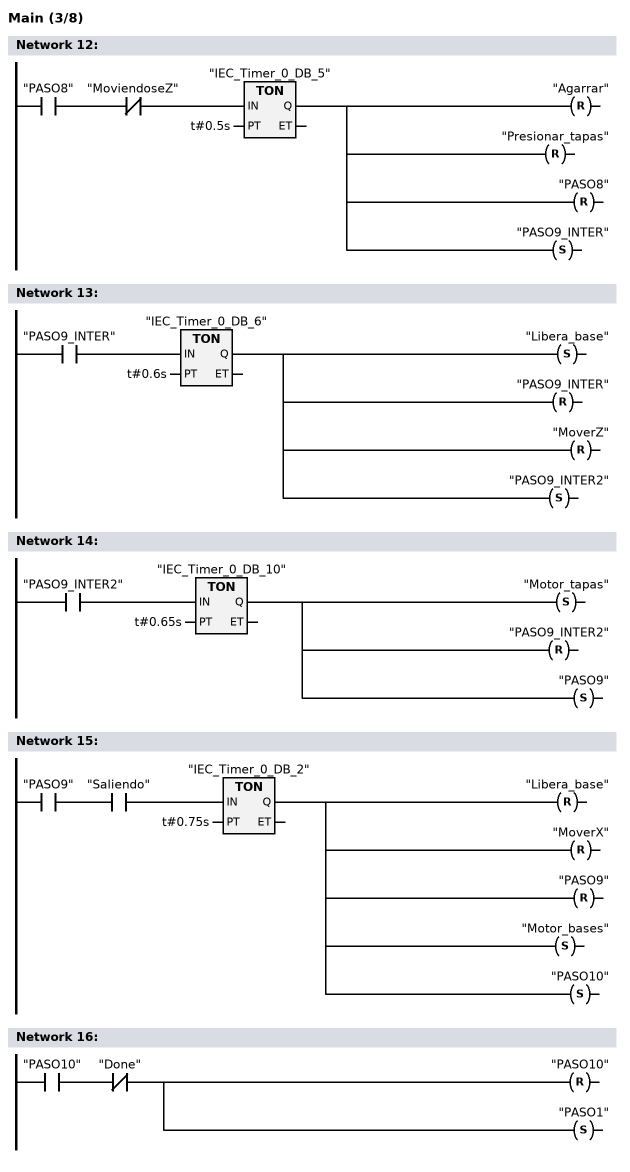
   "IEC_Timer_0_DB_5".TON(IN := "PASO8" AND NOT "MoviendoseZ", PT := t#0.5s);
   IF "IEC_Timer_0_DB_5".Q THEN
       "Agarrar" := FALSE;
       "Presionar_tapas" := FALSE;
       "PASO8" := FALSE;
       "PASO9_INTER" := TRUE;
   END_IF;
END_REGION

REGION Network 13
   "IEC_Timer_0_DB_6".TON(IN := "PASO9_INTER", PT := t#0.6s);
   IF "IEC_Timer_0_DB_6".Q THEN
       "Libera_base" := TRUE;
       "PASO9_INTER" := FALSE;
       "MoverZ" := FALSE;
       "PASO9_INTER2" := TRUE;
   END_IF;
END_REGION

REGION Network 14
   "IEC_Timer_0_DB_10".TON(IN := "PASO9_INTER2", PT := t#0.65s);
   IF "IEC_Timer_0_DB_10".Q THEN
       "Motor_tapas" := TRUE;
       "PASO9_INTER2" := FALSE;
       "PASO9" := TRUE;
   END_IF;
END_REGION

REGION Network 15
   "IEC_Timer_0_DB_2".TON(IN := "PASO9" AND "Saliendo", PT := t#0.75s);
   IF "IEC_Timer_0_DB_2".Q THEN
       "Libera_base" := FALSE;
       "MoverX" := FALSE;
       "PASO9" := FALSE;
       "Motor_bases" := TRUE;
       "PASO10" := TRUE;
   END_IF;
END_REGION

REGION Network 16
   RUNG wire#powerrail
      Contact( "PASO10" )
      I_Contact( "Done" )
      wire#w1
      R_Coil( "PASO10" )
   END_RUNG
   RUNG wire#w1
      S_Coil( "PASO1" )
   END_RUNG
   // the same network as SCL:
   #_w1 := "PASO10" AND NOT "Done";
   IF #_w1 THEN
       "PASO10" := FALSE;
       "PASO1" := TRUE;
   END_IF;
END_REGION

REGION Network 17
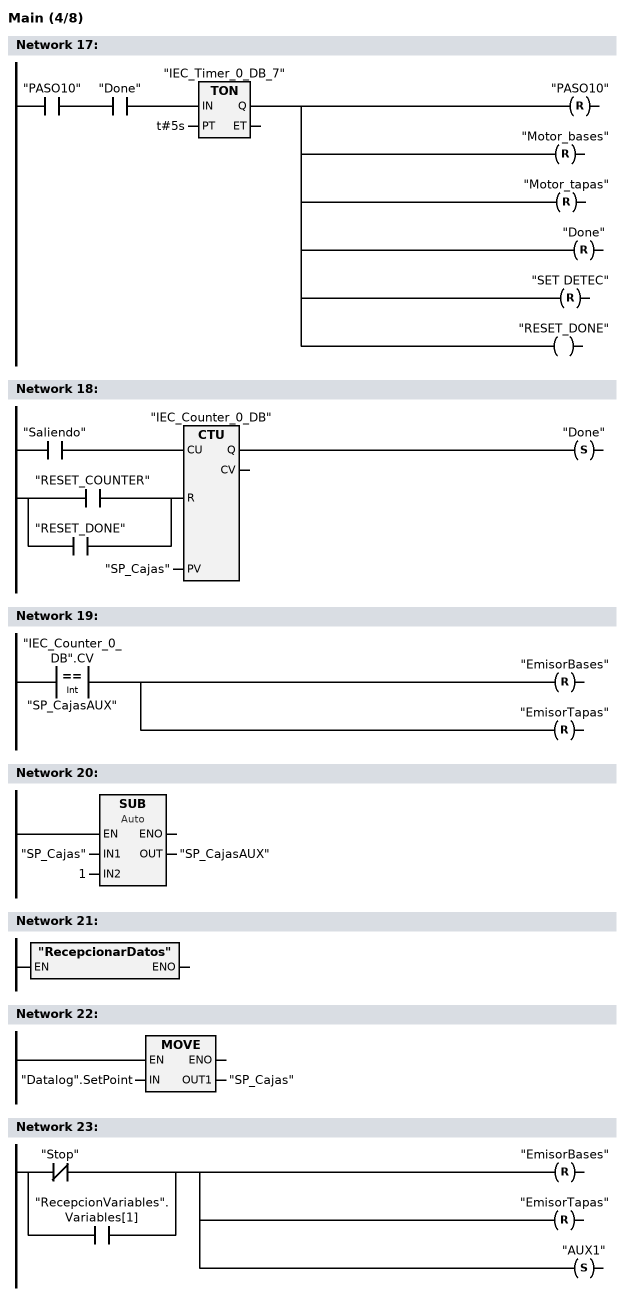
   "IEC_Timer_0_DB_7".TON(IN := "PASO10" AND "Done", PT := t#5s);
   IF "IEC_Timer_0_DB_7".Q THEN
       "PASO10" := FALSE;
       "Motor_bases" := FALSE;
       "Motor_tapas" := FALSE;
       "Done" := FALSE;
       "SET DETEC" := FALSE;
   END_IF;
   "RESET_DONE" := "IEC_Timer_0_DB_7".Q;
END_REGION

REGION Network 18
   "IEC_Counter_0_DB".CTU(CU := "Saliendo", R := "RESET_COUNTER" OR "RESET_DONE", PV := "SP_Cajas");
   IF "IEC_Counter_0_DB".Q THEN "Done" := TRUE; END_IF;
END_REGION

REGION Network 19
   RUNG wire#powerrail
      { S7_Templates := "SrcType := Int" } EQ_Contact(in1 := "IEC_Counter_0_DB".CV, in2 := "SP_CajasAUX")
      wire#w1
      R_Coil( "EmisorBases" )
   END_RUNG
   RUNG wire#w1
      R_Coil( "EmisorTapas" )
   END_RUNG
   // the same network as SCL:
   IF "IEC_Counter_0_DB".CV = "SP_CajasAUX" THEN
       "EmisorBases" := FALSE;
       "EmisorTapas" := FALSE;
   END_IF;
END_REGION

REGION Network 20
   RUNG wire#powerrail
      Sub(in1 := "SP_Cajas", in2 := 1, out => "SP_CajasAUX")
   END_RUNG
   // the same network as SCL:
   "SP_CajasAUX" := "SP_Cajas" - 1;
END_REGION

REGION Network 21
   RUNG wire#powerrail
      "RecepcionarDatos"()
   END_RUNG
   // the same network as SCL:
   "RecepcionarDatos"();
END_REGION

REGION Network 22
   RUNG wire#powerrail
      Move(in := "Datalog".SetPoint, out1 => "SP_Cajas")
   END_RUNG
   // the same network as SCL:
   "SP_Cajas" := "Datalog".SetPoint;
END_REGION

REGION Network 23
   RUNG wire#powerrail
      I_Contact( "Stop" )
      wire#w1
      R_Coil( "EmisorBases" )
   END_RUNG
   RUNG wire#powerrail
      Contact( "RecepcionVariables".Variables[1] )
   END_RUNG wire#w1
   RUNG wire#w1
      R_Coil( "EmisorTapas" )
   END_RUNG
   RUNG wire#w1
      S_Coil( "AUX1" )
   END_RUNG
   // the same network as SCL:
   IF NOT "Stop" OR "RecepcionVariables".Variables[1] THEN
       "EmisorBases" := FALSE;
       "EmisorTapas" := FALSE;
       "AUX1" := TRUE;
   END_IF;
END_REGION

REGION Network 24
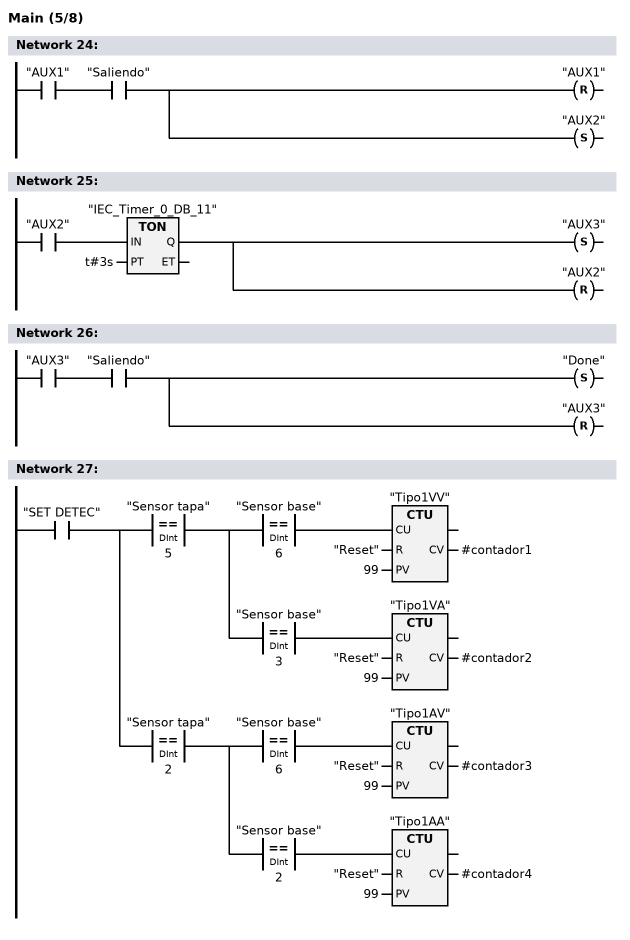
   RUNG wire#powerrail
      Contact( "AUX1" )
      Contact( "Saliendo" )
      wire#w1
      R_Coil( "AUX1" )
   END_RUNG
   RUNG wire#w1
      S_Coil( "AUX2" )
   END_RUNG
   // the same network as SCL:
   #_w1 := "AUX1" AND "Saliendo";
   IF #_w1 THEN
       "AUX1" := FALSE;
       "AUX2" := TRUE;
   END_IF;
END_REGION

REGION Network 25
   "IEC_Timer_0_DB_11".TON(IN := "AUX2", PT := t#3s);
   IF "IEC_Timer_0_DB_11".Q THEN
       "AUX3" := TRUE;
       "AUX2" := FALSE;
   END_IF;
END_REGION

REGION Network 26
   RUNG wire#powerrail
      Contact( "AUX3" )
      Contact( "Saliendo" )
      wire#w1
      S_Coil( "Done" )
   END_RUNG
   RUNG wire#w1
      R_Coil( "AUX3" )
   END_RUNG
   // the same network as SCL:
   IF "AUX3" AND "Saliendo" THEN
       "Done" := TRUE;
       "AUX3" := FALSE;
   END_IF;
END_REGION

REGION Network 27
   #_w1 := "SET DETEC" AND ("Sensor tapa" = 5);
   "Tipo1VV".CTU(CU := #_w1 AND ("Sensor base" = 6), R := "Reset", PV := 99, CV => #contador1);
   "Tipo1VA".CTU(CU := #_w1 AND ("Sensor base" = 3), R := "Reset", PV := 99, CV => #contador2);
   #_w2 := "SET DETEC" AND ("Sensor tapa" = 2);
   "Tipo1AV".CTU(CU := #_w2 AND ("Sensor base" = 6), R := "Reset", PV := 99, CV => #contador3);
   "Tipo1AA".CTU(CU := #_w2 AND ("Sensor base" = 2), R := "Reset", PV := 99, CV => #contador4);
END_REGION

REGION Network 28
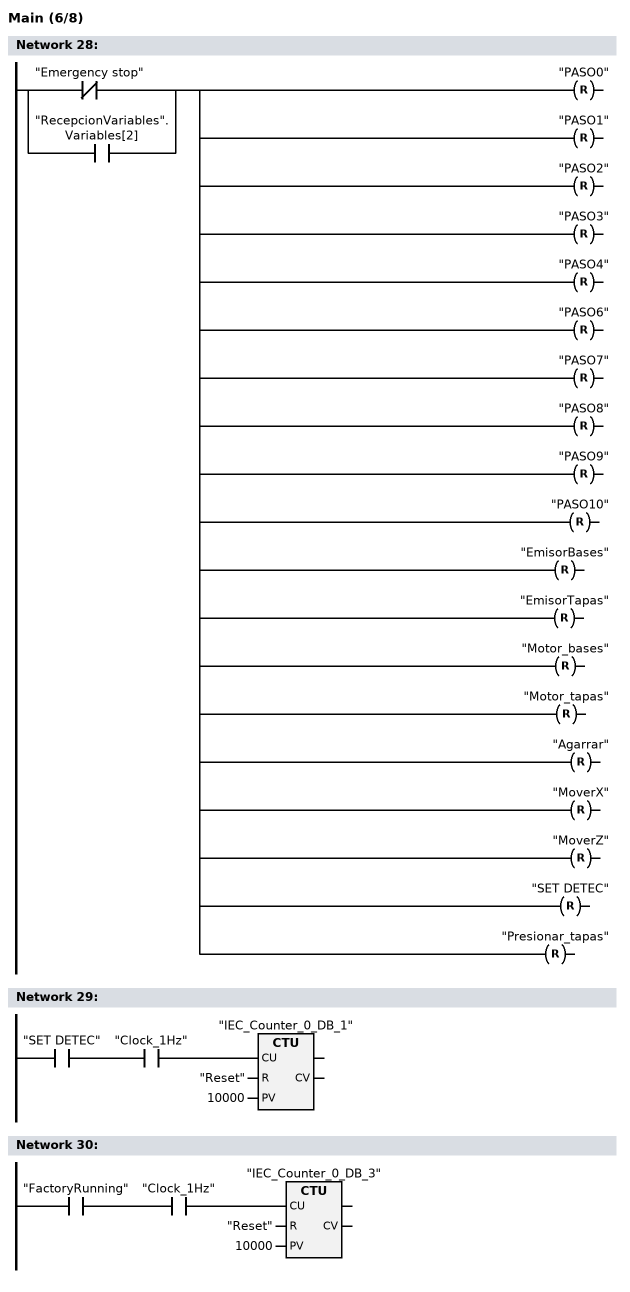
   RUNG wire#powerrail
      I_Contact( "Emergency stop" )
      wire#w1
      R_Coil( "PASO0" )
   END_RUNG
   RUNG wire#powerrail
      Contact( "RecepcionVariables".Variables[2] )
   END_RUNG wire#w1
   RUNG wire#w1
      R_Coil( "PASO1" )
   END_RUNG
   RUNG wire#w1
      R_Coil( "PASO2" )
   END_RUNG
   RUNG wire#w1
      R_Coil( "PASO3" )
   END_RUNG
   RUNG wire#w1
      R_Coil( "PASO4" )
   END_RUNG
   RUNG wire#w1
      R_Coil( "PASO6" )
   END_RUNG
   RUNG wire#w1
      R_Coil( "PASO7" )
   END_RUNG
   RUNG wire#w1
      R_Coil( "PASO8" )
   END_RUNG
   RUNG wire#w1
      R_Coil( "PASO9" )
   END_RUNG
   RUNG wire#w1
      R_Coil( "PASO10" )
   END_RUNG
   RUNG wire#w1
      R_Coil( "EmisorBases" )
   END_RUNG
   RUNG wire#w1
      R_Coil( "EmisorTapas" )
   END_RUNG
   RUNG wire#w1
      R_Coil( "Motor_bases" )
   END_RUNG
   RUNG wire#w1
      R_Coil( "Motor_tapas" )
   END_RUNG
   RUNG wire#w1
      R_Coil( "Agarrar" )
   END_RUNG
   RUNG wire#w1
      R_Coil( "MoverX" )
   END_RUNG
   RUNG wire#w1
      R_Coil( "MoverZ" )
   END_RUNG
   RUNG wire#w1
      R_Coil( "SET DETEC" )
   END_RUNG
   RUNG wire#w1
      R_Coil( "Presionar_tapas" )
   END_RUNG
   // the same network as SCL:
   IF NOT "Emergency stop" OR "RecepcionVariables".Variables[2] THEN
       "PASO0" := FALSE;
       "PASO1" := FALSE;
       "PASO2" := FALSE;
       "PASO3" := FALSE;
       "PASO4" := FALSE;
       "PASO6" := FALSE;
       "PASO7" := FALSE;
       "PASO8" := FALSE;
       "PASO9" := FALSE;
       "PASO10" := FALSE;
       "EmisorBases" := FALSE;
       "EmisorTapas" := FALSE;
       "Motor_bases" := FALSE;
       "Motor_tapas" := FALSE;
       "Agarrar" := FALSE;
       "MoverX" := FALSE;
       "MoverZ" := FALSE;
       "SET DETEC" := FALSE;
       "Presionar_tapas" := FALSE;
   END_IF;
END_REGION

REGION Network 29
   "IEC_Counter_0_DB_1".CTU(CU := "SET DETEC" AND "Clock_1Hz", R := "Reset", PV := 10000);
END_REGION

REGION Network 30
   "IEC_Counter_0_DB_3".CTU(CU := "FactoryRunning" AND "Clock_1Hz", R := "Reset", PV := 10000);
END_REGION

REGION Network 31
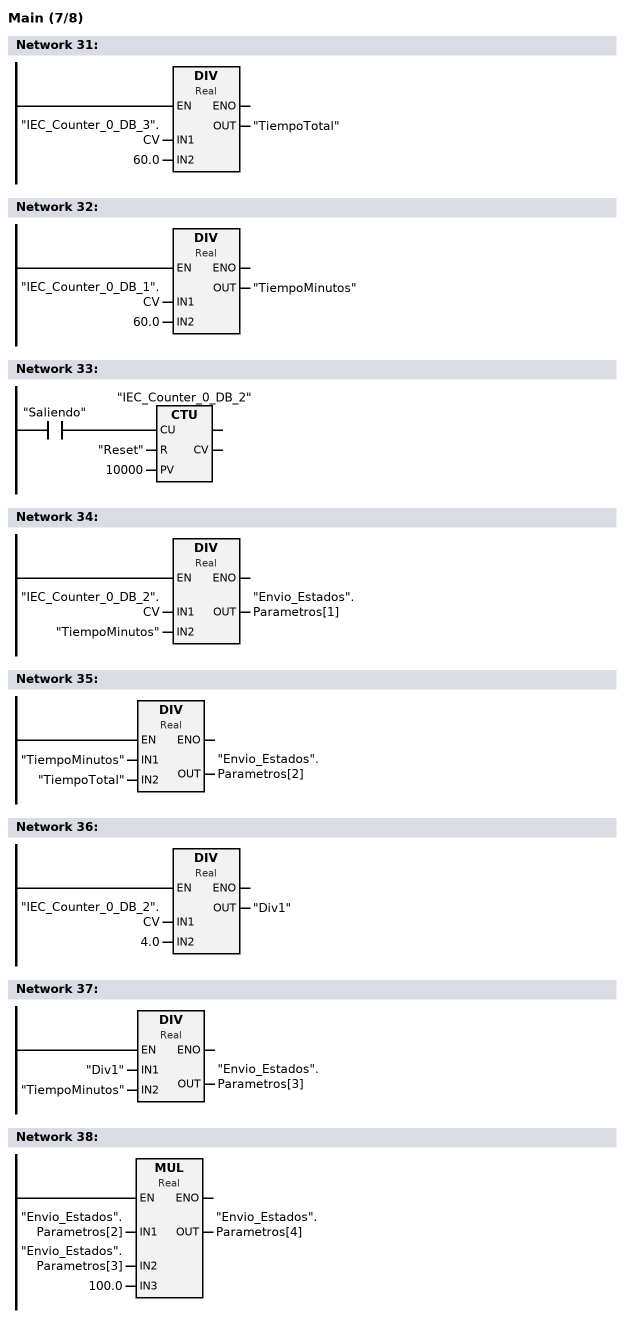
   RUNG wire#powerrail
      { S7_Templates := "SrcType := Real" } Div(in1 := "IEC_Counter_0_DB_3".CV, in2 := 60.0, out => "TiempoTotal")
   END_RUNG
   // the same network as SCL:
   "TiempoTotal" := "IEC_Counter_0_DB_3".CV / 60.0;
END_REGION

REGION Network 32
   RUNG wire#powerrail
      { S7_Templates := "SrcType := Real" } Div(in1 := "IEC_Counter_0_DB_1".CV, in2 := 60.0, out => "TiempoMinutos")
   END_RUNG
   // the same network as SCL:
   "TiempoMinutos" := "IEC_Counter_0_DB_1".CV / 60.0;
END_REGION

REGION Network 33
   "IEC_Counter_0_DB_2".CTU(CU := "Saliendo", R := "Reset", PV := 10000);
END_REGION

REGION Network 34
   RUNG wire#powerrail
      { S7_Templates := "SrcType := Real" } Div(in1 := "IEC_Counter_0_DB_2".CV, in2 := "TiempoMinutos", out => "Envio_Estados".Parametros[1])
   END_RUNG
   // the same network as SCL:
   "Envio_Estados".Parametros[1] := "IEC_Counter_0_DB_2".CV / "TiempoMinutos";
END_REGION

REGION Network 35
   RUNG wire#powerrail
      { S7_Templates := "SrcType := Real" } Div(in1 := "TiempoMinutos", in2 := "TiempoTotal", out => "Envio_Estados".Parametros[2])
   END_RUNG
   // the same network as SCL:
   "Envio_Estados".Parametros[2] := "TiempoMinutos" / "TiempoTotal";
END_REGION

REGION Network 36
   RUNG wire#powerrail
      { S7_Templates := "SrcType := Real" } Div(in1 := "IEC_Counter_0_DB_2".CV, in2 := 4.0, out => "Div1")
   END_RUNG
   // the same network as SCL:
   "Div1" := "IEC_Counter_0_DB_2".CV / 4.0;
END_REGION

REGION Network 37
   RUNG wire#powerrail
      { S7_Templates := "SrcType := Real" } Div(in1 := "Div1", in2 := "TiempoMinutos", out => "Envio_Estados".Parametros[3])
   END_RUNG
   // the same network as SCL:
   "Envio_Estados".Parametros[3] := "Div1" / "TiempoMinutos";
END_REGION

REGION Network 38
   RUNG wire#powerrail
      { S7_Templates := "SrcType := Real" } Mul(in1 := "Envio_Estados".Parametros[2], in2 := "Envio_Estados".Parametros[3], in3 := 100.0, out => "Envio_Estados".Parametros[4])
   END_RUNG
   // the same network as SCL:
   "Envio_Estados".Parametros[4] := "Envio_Estados".Parametros[2] * "Envio_Estados".Parametros[3] * 100.0;
END_REGION

REGION Network 39
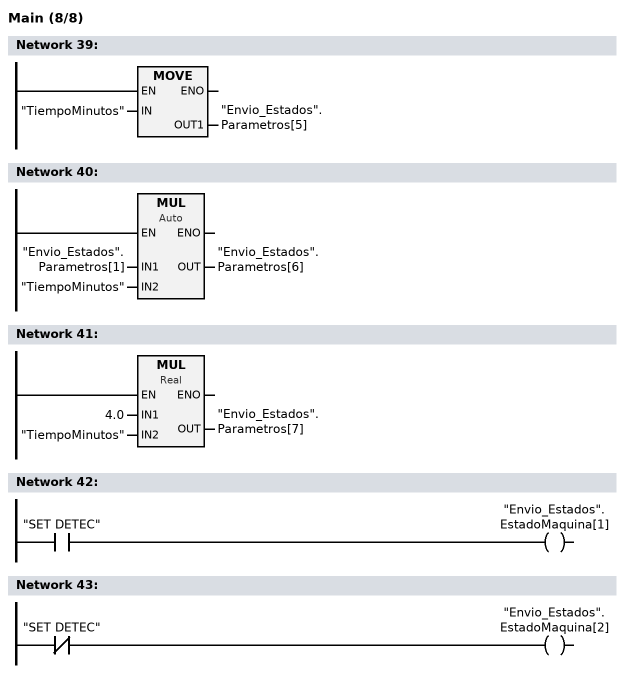
   RUNG wire#powerrail
      Move(in := "TiempoMinutos", out1 => "Envio_Estados".Parametros[5])
   END_RUNG
   // the same network as SCL:
   "Envio_Estados".Parametros[5] := "TiempoMinutos";
END_REGION

REGION Network 40
   RUNG wire#powerrail
      Mul(in1 := "Envio_Estados".Parametros[1], in2 := "TiempoMinutos", out => "Envio_Estados".Parametros[6])
   END_RUNG
   // the same network as SCL:
   "Envio_Estados".Parametros[6] := "Envio_Estados".Parametros[1] * "TiempoMinutos";
END_REGION

REGION Network 41
   RUNG wire#powerrail
      { S7_Templates := "SrcType := Real" } Mul(in1 := 4.0, in2 := "TiempoMinutos", out => "Envio_Estados".Parametros[7])
   END_RUNG
   // the same network as SCL:
   "Envio_Estados".Parametros[7] := 4.0 * "TiempoMinutos";
END_REGION

REGION Network 42
   RUNG wire#powerrail
      Contact( "SET DETEC" )
      Coil( "Envio_Estados".EstadoMaquina[1] )
   END_RUNG
   // the same network as SCL:
   "Envio_Estados".EstadoMaquina[1] := "SET DETEC";
END_REGION

REGION Network 43
   RUNG wire#powerrail
      I_Contact( "SET DETEC" )
      Coil( "Envio_Estados".EstadoMaquina[2] )
   END_RUNG
   // the same network as SCL:
   "Envio_Estados".EstadoMaquina[2] := NOT "SET DETEC";
END_REGION
END_ORGANIZATION_BLOCK

// folder: LGF/4 Math operations

FUNCTION "LGF_RandomRange_Real" : Real   // FC10014, SCL
TITLE = LGF_RandomRange_Real
{ S7_Optimized_Access := 'TRUE' }
AUTHOR : Siemens_Digital_Industries
FAMILY : LGF
NAME : LGF_RandomRange_Real
// This function generates a random value in defined limits with each call.  
// The random number has the data type Real in the specified range.
// Diese Funktion generiert bei jedem Aufruf einen zufälligen Wert zwischen einem definierten Max- und Minwert.  
// Die Zufallszahl hat den Datentyp Real im spezifiziertem Wertebereich.
   VAR_INPUT
      minValue : Real;   // Minimalwert der für den Wertebereich der Zufallszahl - Untergrenze / Minimum value of the range of the random number - lower border
      maxValue : Real;   // Maximalwert der für den Wertebereich der Zufallszahl - Obergrenze / Maximum value of the range of the random number - upper border
   END_VAR
   VAR_OUTPUT
      error : Bool;   // FALSE: No error TRUE: An error occurred during the execution of the FB / FALSE: Kein Fehler TRUE: Während der Ausführung des FB ist ein Fehler aufgetreten
      status : Word;   // 16#0000-16#7FFF: Status of the FB 16#8000-16#FFFF: Error identification (see following Table) / 16#0000-16#7FFF: Status des FB 16#8000-16#FFFF: Fehleridentifikation (siehe folgende Tabelle)
      subfunctionStatus : Word;   // Status or return value of called FB's, FC's and system blocks / Status oder Rückgabewert von aufgerufenen FB's / FC's und Systemfunktionen
   END_VAR
   VAR_TEMP
      tempTime : DTL;   // Temp memory for System time / Temp variable für System Zeit
      tempNanoSecondInDWord : DWord;   // Temp UDInt converted to DWord for access to individual bytes / Temp UDInt konvertiert nach Dword für den Zufriff per Slice auf die Bytes
      tempTimeStatus : Word;   // Temp status of the instruction `RD_SYS_T` / Temp Status der Systemfunktion `RD_SYS_T`
      tempRandomValue : DWord;   // Temp Random startvalue / Temp Zufallswert als Startwert
      tempNormReal : Real;   // Temp normalized Real value (0.0 - 1.0) / Temp Normalisierer Realwert (0.0 - 1.0)
   END_VAR
   // Ret_Val : Random Real number in the predefined range / Zufallszahl vom Datentyp Real im definierten Wertebereich
   VAR CONSTANT
      ZERO : Real := 0.0;   // Zero / 0.0 - value in case of error / Null / 0.0 - Rückgabewert im Fehlerfall
      MAX_UDINT : UDInt := 4294967295;   // Maximum UDInt datatype / Maximalwert eines UDInt Datentype
      SUB_STATUS_NO_ERROR : Word := 16#0000;   // Status: sub function call ends without error / Status: Unterfunktionsaufruf ohne Fehler beendet
      STATUS_FINISHED_NO_ERROR : Word := 16#0000;   // Execution finished without errors / Abarbeitung ohne Fehler beendet
      ERR_MAX_LESS_MIN : Word := 16#8200;   // Error: The ranges specified are wrong: `minValue` is greater than `maxValue` / Fehler: Der spezifizierte Wetebereich is fehlerhaft: `minValue` ist größer als `maxValue`
      ERR_RD_SYS_T : Word := 16#8600;   // Error in `RD_SYS_T` command - check `subFunctionStatus` code / Fehler in Anweisung `RD_SYS_T` - weitere infos in `subFunctionStatus`
   END_VAR
BEGIN
   REGION Block info header
     //=============================================================================
     // SIEMENS AG / (c)Copyright 2017
     //-----------------------------------------------------------------------------
     // Title:            LGF_RandomRange_Real
     // Comment/Function: This function generates random numbers in defined limits (Datatype Real)
     // Library/Family:   LGF(Library General Functions)
     // Author:           Siemens Digital Industry Support
     // Tested with:      S7-PLCSIM Advanced V2.0 SP1
     // Engineering:      TIA Portal V15 Update 2
     // Restrictions:     ENO disabled - error handling done by error and status
     // Requirements:     PLC (S7-1200 / S7-1500)
     //-------------------------------------------------------------------------------
     // Change log table:
     // Version  | Date       | Expert in charge       | Changes applied
     //----------|------------|------------------------|------------------------------
     // 01.00.00 19.08.2015  Siemens Industry Online Support
     //                      First released version
     // 01.00.01 02.01.2017  Siemens Industry Online Support
     //                      Upgrade: TIA Portal V14 Update 1
     // 01.00.02 02.03.2017  Siemens Industry Online Support
     //                      Bugfix: FC number
     // 01.00.03 17.08.2018  Siemens Industry Online Support
     //                      Upgrade: TIA V15 Update 2
     // 01.00.04 23.11.2018  Siemens Industry Online Support
     //                      Upgrade: TIA V15.1
     // 01.01.00 13.11.2019  Simatic Systems Support
     //                      Renamed from "LGF_RandomReal" to "LGF_RandomRange_Real"
     //                      Regions, comments and constants are added
     // 03.00.00 23.04.2020  Simatic Systems Support
     //                      Set version to V3.0.0, harmonize the version of the whole library
     // 03.00.01 04.02.2021  Simatic Systems Support
     //                      Insert documentation
     //=============================================================================
   END_REGION Block info header

   REGION DESCRIPTION
     (/*Note
   :    The status of called commands is output in `subFunctionStatus`. In this case, the output value in `status` indicates which command caused the error. In this case, refer to the TIA Portal Online Help section for information on the respective commands.

   The block generates random values that are between the specified `minValue` and the `maxValue`. This random value is output via the `Ret_Val`.

   The random value is formed from the nanoseconds of the current system time of the CPU. The byte order of this value is inverted and then converted to a floating point.
   Hinweis
   :    In `subFunctionStatus` wird der Status von aufgerufenen Anweisungen ausgegeben. Der Ausgangswert in `status` gibt in diesem Fall an, welche Anweisung den Fehler verursacht hat. Holen Sie sich in diesem Fall die Informationen aus der TIA Portal Online Hilfe zu den jeweiligen Anweisungen.

   Der Baustein generiert zufällige Werte, die zwischen dem angegebenen `minValue`-Wert und `maxValue`-Wert liegen. Dieser zufällige Wert wird über den `Ret_Val` ausgegeben.

   Der Zufallswert wird aus den Nanosekunden der aktuellen Systemzeit der CPU gebildet. Dabei wird die Bytereihenfolge dieses Wertes invertiert und anschließend in eine Gleitkommazahl ungewandelt.*/)
   END_REGION DESCRIPTION

   REGION Validation
     // Check if the maximal Value is less than the minimal value
     IF (#minValue > #maxValue) THEN
       #error := true;
       #status := #ERR_MAX_LESS_MIN;
       #subfunctionStatus := #SUB_STATUS_NO_ERROR;
       #LGF_RandomRange_Real := #ZERO;
       RETURN;
     END_IF;

     // Read system time
     #tempTimeStatus := INT_TO_WORD(RD_SYS_T(#tempTime));

     // Check return variable for error
     IF (#tempTimeStatus <> #SUB_STATUS_NO_ERROR) THEN
       #error := true;
       #status := #ERR_RD_SYS_T;
       #subfunctionStatus := #tempTimeStatus;
       #LGF_RandomRange_Real := #ZERO;
       RETURN;
     END_IF;
   END_REGION

   REGION Calculating random number
     // Converting to double word so individual bytes can be addressed
     #tempNanoSecondInDWord := UDINT_TO_DWORD(#tempTime.NANOSECOND);

     // Calculate a random-start-value depending on the time
     #tempRandomValue.%B3 := #tempNanoSecondInDWord.%B0;
     #tempRandomValue.%B2 := #tempNanoSecondInDWord.%B1;
     #tempRandomValue.%B1 := #tempNanoSecondInDWord.%B2;
     #tempRandomValue.%B0 := #tempNanoSecondInDWord.%B3;

     // Norm the calculated random number: 0.0 <= #tempNormReal <= 1.0
     #tempNormReal := UDINT_TO_REAL(DWORD_TO_UDINT(#tempRandomValue)) / UDINT_TO_REAL(#MAX_UDINT);

     // Scale the tempNormReal to be in the range of maxValue and minValue
     #LGF_RandomRange_Real := ((#tempNormReal * (#maxValue - #minValue) + (#minValue)));

     #error := false;
     #status := #STATUS_FINISHED_NO_ERROR;
     #subfunctionStatus := #SUB_STATUS_NO_ERROR;
     // ENO mechanism is not used
     ENO := TRUE;
   END_REGION
END_FUNCTION